// Mitsubishi GX Works2 project: master   PLC: FX3U/FX3UC

PROGRAM MAIN
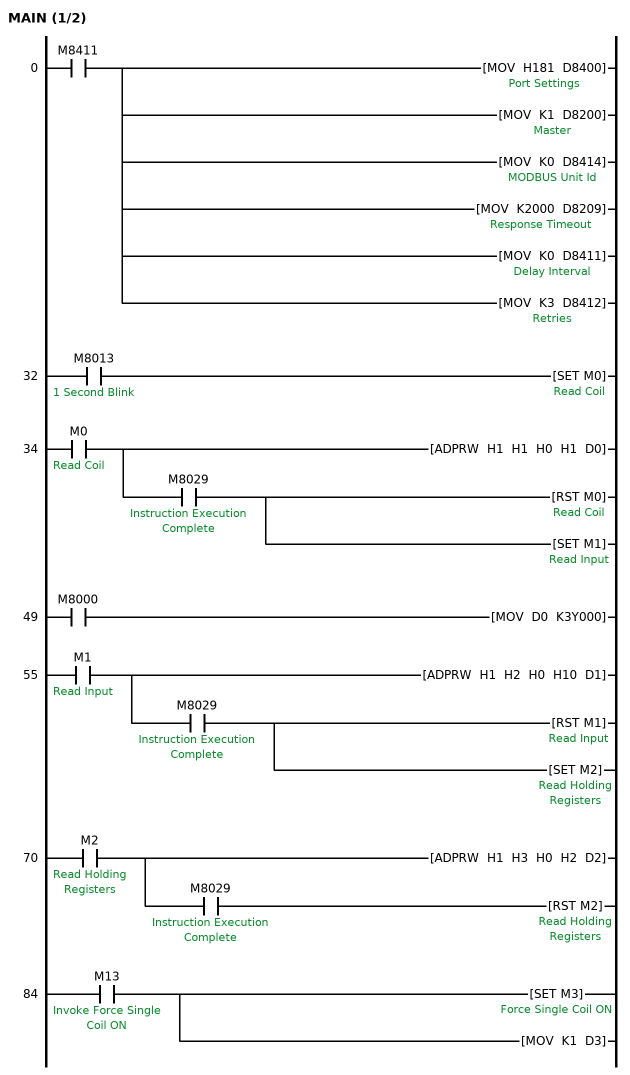
0     LD      M8411
      MOV     H181 D8400  ; Port Settings
      MOV     K1 D8200  ; Master
      MOV     K0 D8414  ; MODBUS Unit Id
      MOV     K2000 D8209  ; Response Timeout
      MOV     K0 D8411  ; Delay Interval
      MOV     K3 D8412  ; Retries
32    LD      M8013  ; 1 Second Blink
      SET     M0  ; Read Coil
34    LD      M0  ; Read Coil
      ADPRW   H1 H1 H0 H1 D0
      AND     M8029  ; Instruction Execution Complete
      RST     M0  ; Read Coil
      SET     M1  ; Read Input
49    LD      M8000
      MOV     D0 K3Y000
55    LD      M1  ; Read Input
      ADPRW   H1 H2 H0 H10 D1
      AND     M8029  ; Instruction Execution Complete
      RST     M1  ; Read Input
      SET     M2  ; Read Holding Registers
70    LD      M2  ; Read Holding Registers
      ADPRW   H1 H3 H0 H2 D2
      AND     M8029  ; Instruction Execution Complete
      RST     M2  ; Read Holding Registers
84    LD      M13  ; Invoke Force Single Coil ON
      SET     M3  ; Force Single Coil ON
      MOV     K1 D3
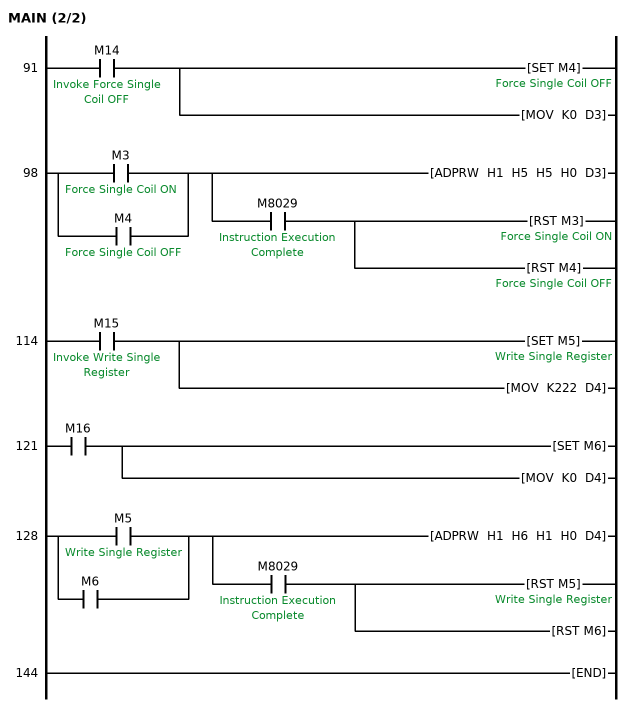
91    LD      M14  ; Invoke Force Single Coil OFF
      SET     M4  ; Force Single Coil OFF
      MOV     K0 D3
98    LD      M3  ; Force Single Coil ON
      OR      M4  ; Force Single Coil OFF
      ADPRW   H1 H5 H5 H0 D3
      AND     M8029  ; Instruction Execution Complete
      RST     M3  ; Force Single Coil ON
      RST     M4  ; Force Single Coil OFF
114   LD      M15  ; Invoke Write Single Register
      SET     M5  ; Write Single Register
      MOV     K222 D4
121   LD      M16
      SET     M6
      MOV     K0 D4
128   LD      M5  ; Write Single Register
      OR      M6
      ADPRW   H1 H6 H1 H0 D4
      AND     M8029  ; Instruction Execution Complete
      RST     M5  ; Write Single Register
      RST     M6
144   END
END_PROGRAM
